(* CoDeSys 2.3.9.50 project: example01pro.pro *)
(* Libraries: STANDARD.LIB 5.6.98 12:03:02, SysLibVisu.lib 7.7.04 18:17:22, SysLibTargetVisu.lib 16.6.08 16:24:26 *)

(* Task configuration *)
TASK Standard (PRIORITY := 0, INTERVAL := T#10ms);
	MAIN
END_TASK
TASK VISU_TASK (PRIORITY := 3, INTERVAL := T#200ms);
	MAINTARGETVISU_PAINT_CODE
END_TASK
TASK VISU_INPUT_TASK (PRIORITY := 2, INTERVAL := T#50ms);
	MAINTARGETVISU_INPUT_CODE
END_TASK

(* Global variable list: Global_Variables *)
VAR_GLOBAL
(*DIGITAL INPUTS*)
	A01_S03_LOCK_BUTTON_NO_DI AT %I* : BOOL;
	A01_S04_PUSH_BUTTON_1_NO_DI AT %I* : BOOL;
	A01_S05_PUSH_BUTTON_2_NO_DI AT %I* : BOOL;
(*DIGITAL OUTPUTS*)
	A01_H01_SIGNAL_LAMP_DO AT %Q* : BOOL;
	A01_K01_MOTOR_RUN_COIL_DO AT %Q* : BOOL;
	A01_K02_MOTOR_DIRECTION_COIL_DO AT %Q* : BOOL;
END_VAR

(* Global variable list: TwinCAT_Configuration *)
(* Generated automatically by TwinCAT - (read only) *)
VAR_CONFIG
	.A01_S03_LOCK_BUTTON_NO_DI AT %IX0.0 : BOOL;
	.A01_S04_PUSH_BUTTON_1_NO_DI AT %IX0.1 : BOOL;
	.A01_S05_PUSH_BUTTON_2_NO_DI AT %IX0.2 : BOOL;
	.A01_H01_SIGNAL_LAMP_DO AT %QX0.0 : BOOL;	(*  ~ {LinkedWith:TIID^Device 1 (EtherCAT)^Term 1 (EK1100)^Term 3 (EL2008)^Channel 1^Output} *)
	.A01_K01_MOTOR_RUN_COIL_DO AT %QX0.1 : BOOL;	(*  ~ {LinkedWith:TIID^Device 1 (EtherCAT)^Term 1 (EK1100)^Term 3 (EL2008)^Channel 2^Output} *)
	.A01_K02_MOTOR_DIRECTION_COIL_DO AT %QX0.2 : BOOL;	(*  ~ {LinkedWith:TIID^Device 1 (EtherCAT)^Term 1 (EK1100)^Term 3 (EL2008)^Channel 3^Output} *)
END_VAR

(* POU MAIN, ST *)
PROGRAM MAIN
VAR
	S3_turned_on:BOOL;
	S4_pushed:BOOL;
	S5_pushed:BOOL;
	motor_runCW:BOOL;
	motor_runCCW:BOOL;
	displayHMI:STRING;
	errorHMI:STRING;
	displayColorHMI:BOOL;
	errorColorHMI:BOOL;
END_VAR
errorHMI:='NO ERRORS';
errorColorHMI:=FALSE;
IF A01_S03_LOCK_BUTTON_NO_DI THEN
	S3_turned_on:=TRUE;
ELSE
	S3_turned_on:=FALSE;
END_IF

IF A01_S04_PUSH_BUTTON_1_NO_DI THEN
	S4_pushed:=TRUE;
ELSE
	S4_pushed:=FALSE;
END_IF

IF A01_S05_PUSH_BUTTON_2_NO_DI THEN
	S5_pushed:=TRUE;
ELSE
	S5_pushed:=FALSE;
END_IF

IF S4_pushed AND NOT S5_pushed THEN
	motor_runCW:=TRUE;
	motor_runCCW:=FALSE;
END_IF

IF S5_pushed AND NOT S4_pushed THEN
	motor_runCCW:=TRUE;
	motor_runCW:=FALSE;
END_IF

IF S4_pushed AND S5_pushed THEN
	motor_runCW:=FALSE;
	motor_runCCW:=FALSE;
	errorHMI:='ONE BUTTON ONLY';
	errorColorHMI:=TRUE;
END_IF

IF NOT S4_pushed AND NOT S5_pushed THEN
	motor_runCW:=FALSE;
	motor_runCCW:=FALSE;
END_IF

IF motor_runCW THEN
	A01_K01_MOTOR_RUN_COIL_DO:=TRUE;
	A01_K02_MOTOR_DIRECTION_COIL_DO:=FALSE;
	displayHMI:='CW';
	displayColorHMI:=TRUE;
	IF S3_turned_on THEN
		A01_H01_SIGNAL_LAMP_DO:=TRUE;
	ELSE
		A01_H01_SIGNAL_LAMP_DO:=FALSE;
	END_IF
END_IF

IF motor_runCCW THEN
	A01_K01_MOTOR_RUN_COIL_DO:=TRUE;
	A01_K02_MOTOR_DIRECTION_COIL_DO:=TRUE;
	displayHMI:='CCW';
	displayColorHMI:=TRUE;
	IF S3_turned_on THEN
		A01_H01_SIGNAL_LAMP_DO:=TRUE;
	ELSE
		A01_H01_SIGNAL_LAMP_DO:=FALSE;
	END_IF
END_IF

IF NOT motor_runCCW AND NOT motor_runCW THEN
	displayHMI:='CW OR CCW?';
	displayColorHMI:=FALSE;
	A01_K01_MOTOR_RUN_COIL_DO:=FALSE;
	A01_K02_MOTOR_DIRECTION_COIL_DO:=FALSE;
	A01_H01_SIGNAL_LAMP_DO:=FALSE;
END_IF
END_PROGRAM

(* Visualisation HMI
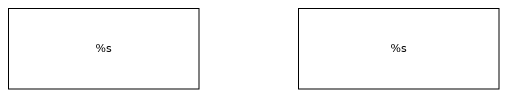
rectangle at (70,150)-(261,231): text "%s"; shows MAIN.displayHMI; alarm colour if MAIN.displayColorHMI
rectangle at (360,150)-(561,231): text "%s"; shows MAIN.errorHMI; alarm colour if MAIN.errorColorHMI
*)
